Staubli VAL3: remSetIP.pgx

program remSetIP(string& sArgs[] (dimensions=1), string& sReturn[] (dimensions=1))
  local bool bOk
  local num nIP
begin
  // Pick the active IP, 0 or 1.
  //
  logMsg("call remSetIP with args "+sArgs)
  toNum(left(sArgs,1),nIP,bOk)
  if bOk
    if nIP==0
      nIPNumber=0
    else
      nIPNumber=1
    endIf
    sReturn="SETIP "+toString("",nIPNumber)
  else
    call remErrNum("SETIP",sArgs,sReturn)
  endIf
end
